FUNCTION_BLOCK StoppableEntity IMPLEMENTS I_Callable
VAR_INPUT
END_VAR
VAR_OUTPUT
END_VAR
VAR
	_ett: EntityStart;
		_onSafetyStop: Receiver := (Callable := THIS^);
	_ettEnd: EntityEnd;

	_bSafetyStopLock: BOOL;
END_VAR

(*
This method provides a standardized way for other objects to interact with the object that owns it.
*)
METHOD Call
VAR_INPUT
	iArg	: StageCore.I_Arg;
END_VAR
VAR
	iSafetyStopState: I_BoolArg;
END_VAR
IF IsOk(IArgToIBoolArg(iArg, iSafetyStopState)) THEN
	_bSafetyStopLock := iSafetyStopState.Get;
END_IF
END_METHOD

END_FUNCTION_BLOCK

(* stored: Version 1.1.0.1
   POU StoppableEntity: Id {a83a5099-ac3d-408e-9581-4d71a7e0c014}, SpecialFunc None
   Method Call: Id {5e277143-6260-438e-8a8a-6388f95da339} *)
